// TIA Portal project "Schema_n1" (V16)
// Progetto schema numero 1.
// Programmazione LADDER

(* hardware
DEVICE "S7-1200 station_1"  S7-1200 Station
   slot 0: "Telaio di montaggio_0"  S7-1200 Rack  Rack  V1.0
   slot 1: "PLC_1"  CPU 1215C DC/DC/Rly  6ES7 215-1HG40-0XB0  V4.4
*)

// ===== PLC "PLC_1"  CPU 1215C DC/DC/Rly =====

VAR_GLOBAL   // PLC tag table "Tabella delle variabili standard"
   "Pulsante di avvio (S1)" AT %I0.0 : Bool;
   "Pulsante di arresto (S2)" AT %I0.1 : Bool;
   "Contatore avvio motore (Q)" AT %Q0.0 : Bool;
END_VAR

ORGANIZATION_BLOCK "Main"   // OB1, LAD, ProgramCycle
TITLE = "Main Program Sweep (Cycle)"
{ S7_Optimized_Access := 'TRUE' }
VERSION : 0.1
   VAR_INPUT
      Initial_Call : Bool;   // Initial call of this OB
      Remanence : Bool;   // =True, if remanent data are available
   END_VAR
BEGIN

REGION Network 1
   // Se viene premuto il pulsante s1 si avvia il contatore quindi il motore viene azionato, alla pressione del pulsante di arresto spengo tutto (se io rilascio il pulsante di arresto il contatore continua a funzionare perchè ho fatto il collegamento di autoritenuta)
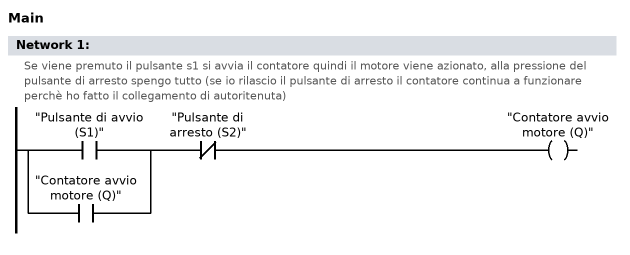
   RUNG wire#powerrail
      Contact( "Pulsante di avvio (S1)" )
      wire#w1
      I_Contact( "Pulsante di arresto (S2)" )
      Coil( "Contatore avvio motore (Q)" )
   END_RUNG
   RUNG wire#powerrail
      Contact( "Contatore avvio motore (Q)" )
   END_RUNG wire#w1
   // the same network as SCL:
   "Contatore avvio motore (Q)" := ("Pulsante di avvio (S1)" OR "Contatore avvio motore (Q)") AND NOT "Pulsante di arresto (S2)";
END_REGION
END_ORGANIZATION_BLOCK